(* LS Electric XG5000 project: 사거리신호등 *)
(* PLC LSPLC *)
VAR_GLOBAL
    four_flash : TIME;
    green_four_time : TIME;
    green_one_time : TIME;
    green_three_time : TIME;
    green_two_time : TIME;
    one_flash : TIME;
    three_flash : TIME;
    two_flash : TIME;
END_VAR

FUNCTION_BLOCK 카운트
VAR_INPUT
    trigger : BOOL;
    남은시간 : TIME;
    전체시간 : TIME;
END_VAR
VAR_OUTPUT
    시간표시 : INT;
END_VAR
VAR
    one_time : INT;
    var2_int : INT;
    var2_udint : UDINT;
    var_int : INT;
    var_udint : UDINT;
    남은시간숫자 : INT;
    전체시간숫자 : INT;
END_VAR

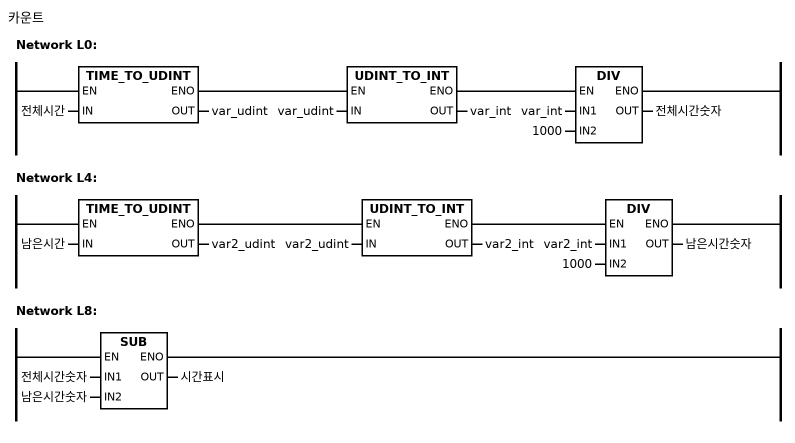
(* Rung L0 *)
var_udint := TIME_TO_UDINT(전체시간);
var_int := UDINT_TO_INT(var_udint);
전체시간숫자 := var_int / 1000;
(* Rung L4 *)
var2_udint := TIME_TO_UDINT(남은시간);
var2_int := UDINT_TO_INT(var2_udint);
남은시간숫자 := var2_int / 1000;
(* Rung L8 *)
시간표시 := 전체시간숫자 - 남은시간숫자;
END_FUNCTION_BLOCK

FUNCTION_BLOCK 사거리신호등
VAR_INPUT
    trigger : BOOL;
END_VAR
VAR
    four_flash : TIME;
    four_green : DWORD := 9054286;
    four_yellow : DWORD := 9054354;
    green_four_time : TIME;
    green_one_time : TIME;
    green_three_time : TIME;
    green_two_time : TIME;
    lamp : BOOL;
    one_flash : TIME;
    one_green : DWORD := 3811489;
    one_yellow : DWORD := 4860066;
    three_flash : TIME;
    three_green : DWORD := 9048994;
    three_yellow : DWORD := 9053346;
    time_four_flash : TON;
    time_four_green : TON;
    time_four_yellow : TON;
    time_one_flash : TON;
    time_one_green : TON;
    time_one_yellow : TON;
    time_three_flash : TON;
    time_three_green : TON;
    time_three_yellow : TON;
    time_two_flash : TON;
    time_two_green : TON;
    time_two_yellow : TON;
    two_flash : TIME;
    two_green : DWORD := 8710306;
    two_yellow : DWORD := 8988834;
    yellow_time : TIME;
END_VAR

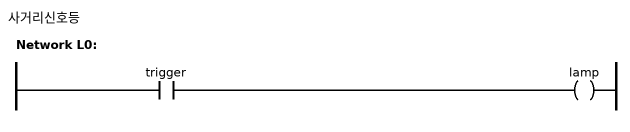
(* Rung L0 *)
lamp := trigger;
END_FUNCTION_BLOCK

FUNCTION_BLOCK 시간변경
VAR_INPUT
    pulse : BOOL;
    change_time_one : TIME;
    change_time_two : TIME;
    change_time_three : TIME;
    change_time_four : TIME;
    change_time_five : TIME;
END_VAR
VAR_OUTPUT
    시간1 : TIME;
    시간2 : TIME;
    시간3 : TIME;
    시간4 : TIME;
    시간5 : TIME;
END_VAR
VAR
    zero : DWORD := 0;
END_VAR

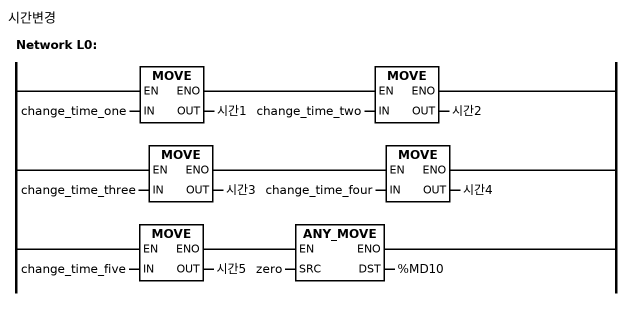
(* Rung L0 *)
시간1 := change_time_one;
시간2 := change_time_two;
시간3 := change_time_three;
시간4 := change_time_four;
시간5 := change_time_five;
%MD10 := ANY_MOVE(SRC := zero);
END_FUNCTION_BLOCK

FUNCTION_BLOCK 메모리시퀀스
VAR_INPUT
    green_memory : DWORD;
    yellow_memory : DWORD;
    time_before : BOOL;
    time_green : BOOL;
    time_flash : BOOL;
    time_yellow : BOOL;
END_VAR
VAR_OUTPUT
    green_light : BOOL;
END_VAR

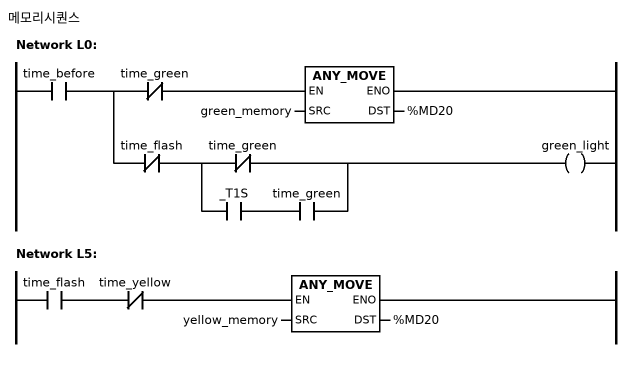
(* Rung L0 *)
IF time_before AND NOT time_green THEN %MD20 := ANY_MOVE(SRC := green_memory); END_IF;
green_light := time_before AND NOT time_flash AND (NOT time_green OR (_T1S AND time_green));
(* Rung L5 *)
IF time_flash AND NOT time_yellow THEN %MD20 := ANY_MOVE(SRC := yellow_memory); END_IF;
END_FUNCTION_BLOCK

FUNCTION_BLOCK 사거리신호등_카운트
VAR_INPUT
    time1 : BOOL;
    time2 : BOOL;
    time3 : BOOL;
    time4 : BOOL;
END_VAR
VAR_EXTERNAL
    four_flash : TIME;
    green_four_time : TIME;
    green_one_time : TIME;
    green_three_time : TIME;
    green_two_time : TIME;
    one_flash : TIME;
    three_flash : TIME;
    two_flash : TIME;
END_VAR
VAR
    카운트1 : 카운트;
    카운트2 : 카운트;
    카운트3 : 카운트;
    카운트4 : 카운트;
END_VAR

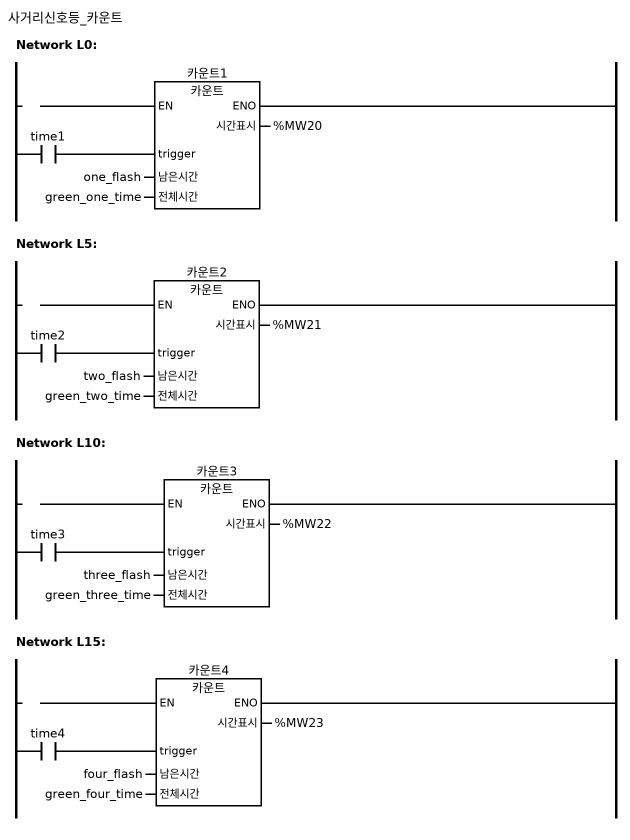
(* Rung L0 *)
(* never executed: 카운트1(trigger := time1, 남은시간 := one_flash, 전체시간 := green_one_time, 시간표시 => %MW20); *)
(* Rung L5 *)
(* never executed: 카운트2(trigger := time2, 남은시간 := two_flash, 전체시간 := green_two_time, 시간표시 => %MW21); *)
(* Rung L10 *)
(* never executed: 카운트3(trigger := time3, 남은시간 := three_flash, 전체시간 := green_three_time, 시간표시 => %MW22); *)
(* Rung L15 *)
(* never executed: 카운트4(trigger := time4, 남은시간 := four_flash, 전체시간 := green_four_time, 시간표시 => %MW23); *)
END_FUNCTION_BLOCK

FUNCTION_BLOCK 사거리신호등_시간변경
VAR_INPUT
    trigger2 : BOOL;
END_VAR
VAR_EXTERNAL
    green_four_time : TIME;
    green_one_time : TIME;
    green_three_time : TIME;
    green_two_time : TIME;
    yellow_time : TIME;
END_VAR
VAR
    도로1번 : 시간변경;
    도로2번 : 시간변경;
    도로3번 : 시간변경;
    도로4번 : 시간변경;
    평상시 : 시간변경;
END_VAR

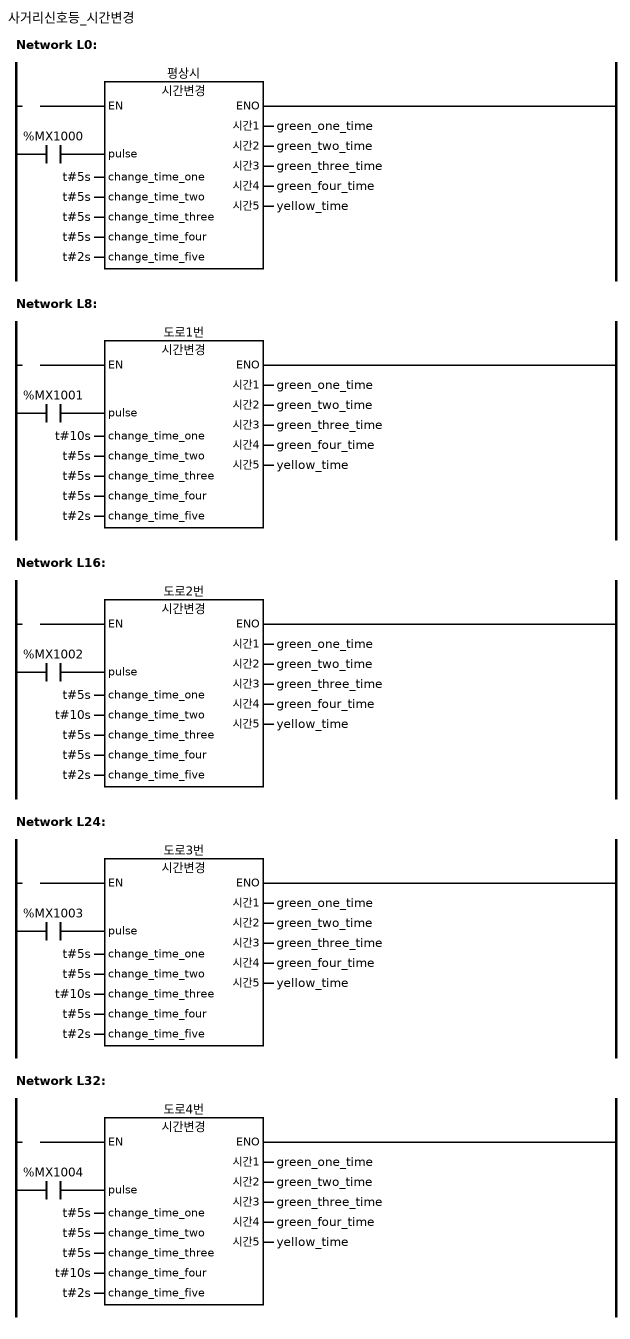
(* Rung L0 *)
(* never executed: 평상시(pulse := %MX1000, change_time_one := t#5s, change_time_two := t#5s, change_time_three := t#5s, change_time_four := t#5s, change_time_five := t#2s, 시간1 => green_one_time, 시간2 => green_two_time, 시간3 => green_three_time, 시간4 => green_four_time, 시간5 => yellow_time); *)
(* Rung L8 *)
(* never executed: 도로1번(pulse := %MX1001, change_time_one := t#10s, change_time_two := t#5s, change_time_three := t#5s, change_time_four := t#5s, change_time_five := t#2s, 시간1 => green_one_time, 시간2 => green_two_time, 시간3 => green_three_time, 시간4 => green_four_time, 시간5 => yellow_time); *)
(* Rung L16 *)
(* never executed: 도로2번(pulse := %MX1002, change_time_one := t#5s, change_time_two := t#10s, change_time_three := t#5s, change_time_four := t#5s, change_time_five := t#2s, 시간1 => green_one_time, 시간2 => green_two_time, 시간3 => green_three_time, 시간4 => green_four_time, 시간5 => yellow_time); *)
(* Rung L24 *)
(* never executed: 도로3번(pulse := %MX1003, change_time_one := t#5s, change_time_two := t#5s, change_time_three := t#10s, change_time_four := t#5s, change_time_five := t#2s, 시간1 => green_one_time, 시간2 => green_two_time, 시간3 => green_three_time, 시간4 => green_four_time, 시간5 => yellow_time); *)
(* Rung L32 *)
(* never executed: 도로4번(pulse := %MX1004, change_time_one := t#5s, change_time_two := t#5s, change_time_three := t#5s, change_time_four := t#10s, change_time_five := t#2s, 시간1 => green_one_time, 시간2 => green_two_time, 시간3 => green_three_time, 시간4 => green_four_time, 시간5 => yellow_time); *)
END_FUNCTION_BLOCK

PROGRAM CodingonProject (* task: 스캔 프로그램 *)
VAR
    change_time : 사거리신호등_시간변경;
    count : 사거리신호등_카운트;
    four_green : DWORD := 9054286;
    four_yellow : DWORD := 9054354;
    memory1 : 메모리시퀀스;
    memory2 : 메모리시퀀스;
    memory3 : 메모리시퀀스;
    memory4 : 메모리시퀀스;
    one_green : DWORD := 3811489;
    one_yellow : DWORD := 4860066;
    three_green : DWORD := 9048994;
    three_yellow : DWORD := 9053346;
    time_four_flash : TON;
    time_four_green : TON;
    time_four_yellow : TON;
    time_one_flash : TON;
    time_one_green : TON;
    time_one_yellow : TON;
    time_three_flash : TON;
    time_three_green : TON;
    time_three_yellow : TON;
    time_two_flash : TON;
    time_two_green : TON;
    time_two_yellow : TON;
    two_green : DWORD := 8710306;
    two_yellow : DWORD := 8988834;
END_VAR
VAR_EXTERNAL
    four_flash : TIME;
    green_four_time : TIME;
    green_one_time : TIME;
    green_three_time : TIME;
    green_two_time : TIME;
    one_flash : TIME;
    three_flash : TIME;
    two_flash : TIME;
    yellow_time : TIME;
END_VAR

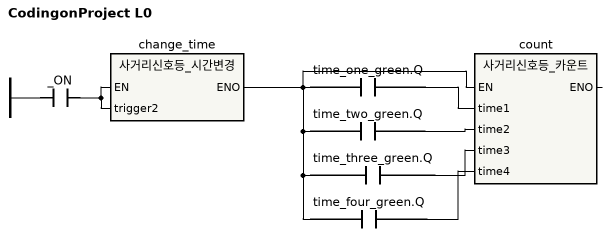
(* Rung L0 *)
IF _ON THEN
    change_time(trigger2 := _ON);
    count(time1 := _ON AND time_one_green.Q, time2 := _ON AND time_two_green.Q, time3 := _ON AND time_three_green.Q, time4 := _ON AND time_four_green.Q);
END_IF;

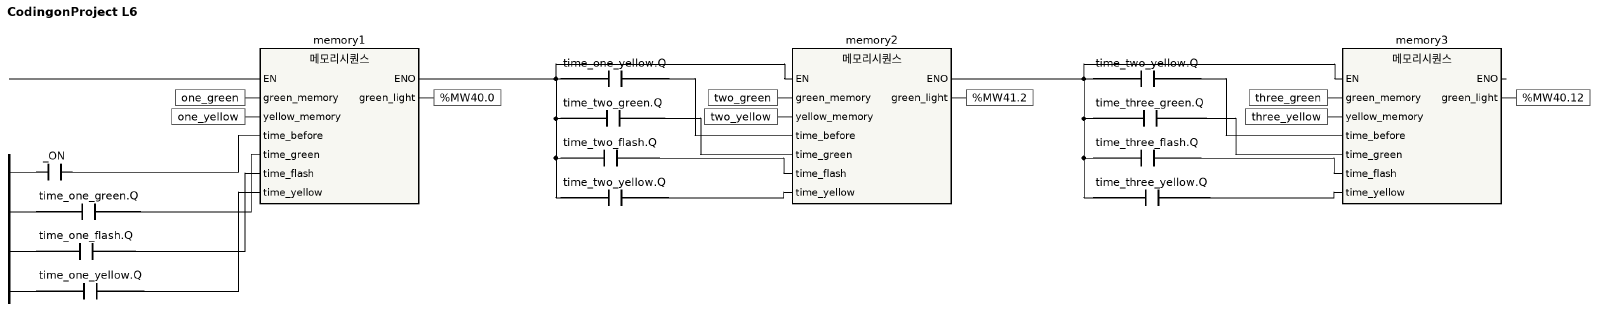
(* Rung L6 *)
memory1(green_memory := one_green, yellow_memory := one_yellow, time_before := _ON, time_green := time_one_green.Q, time_flash := time_one_flash.Q, time_yellow := time_one_yellow.Q);
%MW40.0 := memory1.green_light;
memory2(green_memory := two_green, yellow_memory := two_yellow, time_before := time_one_yellow.Q, time_green := time_two_green.Q, time_flash := time_two_flash.Q, time_yellow := time_two_yellow.Q);
%MW41.2 := memory2.green_light;
memory3(green_memory := three_green, yellow_memory := three_yellow, time_before := time_two_yellow.Q, time_green := time_three_green.Q, time_flash := time_three_flash.Q, time_yellow := time_three_yellow.Q);
%MW40.12 := memory3.green_light;

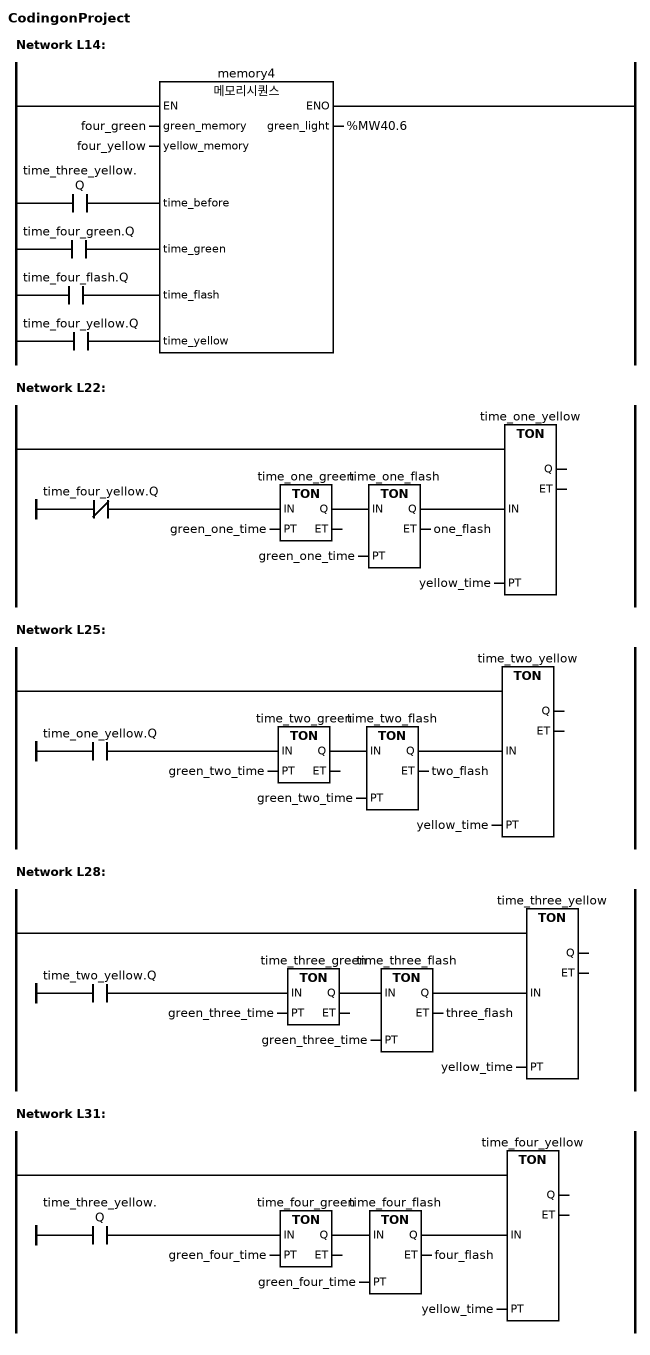
(* Rung L14 *)
memory4(green_memory := four_green, yellow_memory := four_yellow, time_before := time_three_yellow.Q, time_green := time_four_green.Q, time_flash := time_four_flash.Q, time_yellow := time_four_yellow.Q, green_light => %MW40.6);
(* Rung L22 *)
time_one_green(IN := NOT time_four_yellow.Q, PT := green_one_time);
time_one_flash(IN := time_one_green.Q, PT := green_one_time, ET => one_flash);
time_one_yellow(IN := time_one_flash.Q, PT := yellow_time);
(* Rung L25 *)
time_two_green(IN := time_one_yellow.Q, PT := green_two_time);
time_two_flash(IN := time_two_green.Q, PT := green_two_time, ET => two_flash);
time_two_yellow(IN := time_two_flash.Q, PT := yellow_time);
(* Rung L28 *)
time_three_green(IN := time_two_yellow.Q, PT := green_three_time);
time_three_flash(IN := time_three_green.Q, PT := green_three_time, ET => three_flash);
time_three_yellow(IN := time_three_flash.Q, PT := yellow_time);
(* Rung L31 *)
time_four_green(IN := time_three_yellow.Q, PT := green_four_time);
time_four_flash(IN := time_four_green.Q, PT := green_four_time, ET => four_flash);
time_four_yellow(IN := time_four_flash.Q, PT := yellow_time);
END_PROGRAM